// TIA Portal V16 export
// export: Created 2022-07-21T09:35:27.6988541Z, ExportSetting WithDefaults, DisplayName Totally Integrated Automation Portal, DisplayVersion V16 Update 4, DisplayName TIA Portal Version Control Interface, DisplayVersion V16 Update 2, DisplayName TIA Portal Openness, DisplayVersion V16 Update 4, DisplayName SINAMICS Startdrive Advanced, DisplayVersion V16 Update 5, DisplayName SINAMICS Startdrive G130, G150, S120, S150, SINAMICS MV, S210, DisplayVersion V16 Update 5, DisplayName SINAMICS Startdrive G110M, G120, G120C, G120D, G120P, G115D, DisplayVersion V16 Update 5, DisplayName STEP 7 Professional, DisplayVersion V16 Update 4, DisplayName STEP 7 Safety, DisplayVersion V16, DisplayName WinCC Advanced, DisplayVersion V16 Update 4
FUNCTION_BLOCK "lbMeasureAvgCapacity"   // FB111, LAD
TITLE = Measure average capacity / Pomiar średniej wydajności
{ S7_Optimized_Access := 'TRUE' }
VERSION : 0.1
// stored: AutoNumber true, IsIECCheckEnabled true, IsRetainMemResEnabled false, MemoryReserve 100, SetENOAutomatically false, UDAEnableTagReadback false
   VAR_INPUT
      inEnable { ExternalAccessible := 'False'; ExternalVisible := 'False'; ExternalWritable := 'False'} : Bool;   // General release for this object / Generelle Freigabe für das Objekt
      inRENewTU { ExternalAccessible := 'False'; ExternalVisible := 'False'; ExternalWritable := 'False'} : Bool;   // [RE] New TU detected, count +1 / [PF] Neue TE erkannt, zähle +1
      inTimePeriod { ExternalAccessible := 'False'; ExternalVisible := 'False'; ExternalWritable := 'False'} : Time;   // Timeperiod for capacity / Zeitraum für Leistung
      inTimeBaseIntervall : Time := T#1000ms;   // Timebase for intervall
   END_VAR
   VAR_OUTPUT
      ouCapacity { ExternalAccessible := 'False'; ExternalVisible := 'False'; ExternalWritable := 'False'} : UInt;   // Capacity in period of time / Leistung in Zeitraum
      ouCapacitiyHeadToHead { ExternalAccessible := 'False'; ExternalVisible := 'False'; ExternalWritable := 'False'} : UInt;   // Capacity head to head / Leistung Vorderkante zu Vorderkante
      ouTimeHeadToHead { ExternalAccessible := 'False'; ExternalVisible := 'False'; ExternalWritable := 'False'} : Time;   // Time head to head / Zeit Vorderkante zu Vorderkante
   END_VAR
   VAR
      sMeasureAvgCapacityCount { ExternalAccessible := 'False'; ExternalVisible := 'False'; ExternalWritable := 'False'; S7_SetPoint := 'True'} : "fbMeasureAvgCapacityCount";
      sMeasureAvgCapacityGet { ExternalAccessible := 'False'; ExternalVisible := 'False'; ExternalWritable := 'False'; S7_SetPoint := 'True'} : "fbMeasureAvgCapacityGet";
      sBuffer { ExternalAccessible := 'False'; ExternalVisible := 'False'; ExternalWritable := 'False'} : "typeBufferCountTUs";   // Buffer Count TUs / Puffer zum TUs zählen
   END_VAR
BEGIN

REGION Network 1: Call: MeasureAvgCapacity / Wywołanie: MeasureAvgCapacity
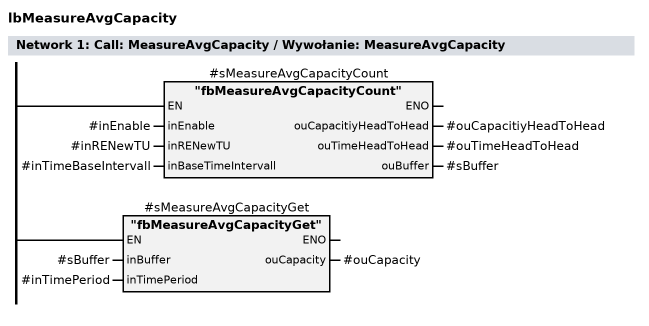
   RUNG wire#powerrail
      #sMeasureAvgCapacityCount(inEnable := #inEnable, inRENewTU := #inRENewTU, inBaseTimeIntervall := #inTimeBaseIntervall, ouCapacitiyHeadToHead => #ouCapacitiyHeadToHead, ouTimeHeadToHead => #ouTimeHeadToHead, ouBuffer => #sBuffer)
   END_RUNG
   RUNG wire#powerrail
      #sMeasureAvgCapacityGet(inBuffer := #sBuffer, inTimePeriod := #inTimePeriod, ouCapacity => #ouCapacity)
   END_RUNG
   // the same network as SCL:
   #sMeasureAvgCapacityCount(inEnable := #inEnable,   // "fbMeasureAvgCapacityCount"
                           inRENewTU := #inRENewTU,
                           inBaseTimeIntervall := #inTimeBaseIntervall,
                           ouCapacitiyHeadToHead => #ouCapacitiyHeadToHead,
                           ouTimeHeadToHead => #ouTimeHeadToHead,
                           ouBuffer => #sBuffer);
   #sMeasureAvgCapacityGet(inBuffer := #sBuffer, inTimePeriod := #inTimePeriod, ouCapacity => #ouCapacity);   // "fbMeasureAvgCapacityGet"
END_REGION
END_FUNCTION_BLOCK
